(* Logix 5000 project; controller Program_Dampproduktion Emulate 5570 rev 32.11; software revision 32.02 *)

TASK MainTask (continuous, watchdog 500 ms) : Simulering
TASK Regulatorer (periodic, rate 100 ms, priority 10, watchdog 500 ms) : Regulator, Damp_Ventil_Regulering

MODULES
   Local : Emulate 5570 (ICP 3, rev 32.11)
END_MODULES

ADD_ON_INSTRUCTION Add_three_Numbers   (* revision 1.0 *)
VAR_INPUT
   nr1 : REAL; {required}
   nr2 : REAL; {required}
   nr3 : REAL; {required}
END_VAR
VAR_OUTPUT
   nr4 : REAL; {access Read Only, required}
END_VAR
VAR
   ADD_01 : FBD_MATH; {access None}
   ADD_02 : FBD_MATH; {access None}
   __lCF223809C1E0D70E : REAL; {access None}
   __l2841EC67DFDD29AE : REAL; {access None}
   __l253A293BB21A6975 : REAL; {access None}
END_VAR

ROUTINE Logic   (* function block diagram *)
   SHEET 1
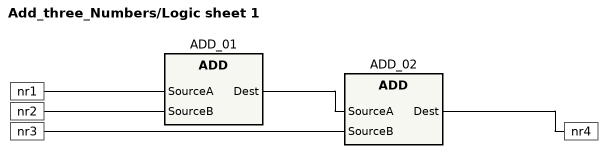
   ADD_01 : ADD(SourceA := nr1, SourceB := nr2);
   ADD_02 : ADD(SourceA := ADD_01.Dest, SourceB := nr3);
   nr4 := ADD_02.Dest;
END_ROUTINE
END_ADD_ON_INSTRUCTION

ADD_ON_INSTRUCTION DampProces   (* revision 1.0, vendor JPJohansen  *)
// Til obligatorisk opgave 1 - PA3
// Revision note:
// ændringer på dødtid og tidskonstant samt navn. den
VAR_INPUT
   belastning : REAL;
   DeadTime : REAL := 2.0;   // Dødtid 0.1 til 1.99 sek.
   Tidskonstant : REAL := 20.0;   // Tidskonstant i LeadLag 0.1 til 40.0 sek
END_VAR
VAR_OUTPUT
   PV : REAL; {access Read Only, required}
END_VAR
VAR_INPUT
   CV : REAL; {required}
END_VAR
VAR
   DEDT_01 : DEADTIME := (Deadtime := 1.0, Gain := 1.0, RTSTime := 1);
   ADD_01 : FBD_MATH;
   LDLG_01 : LEAD_LAG := (Lag := 20.0, Gain := 1.0, RTSTime := 1);
   HLL_01 : HL_LIMIT := (HighLimit := 100.0);
   SCL_01 : SCALE := (InRawMax := 100.0, InEUMax := 15.0, Limiting := 1); {access None}
   SCL_02 : SCALE := (InRawMax := 100.0, InEUMax := -100.0, Limiting := 1); {access None}
   StorageA : REAL[200]; {access None}
   SCL_03 : SCALE := (InRawMax := 100.0, InEUMin := 100.0, Limiting := 1); {access None}
   __lBFE748FCFA657C66 : REAL; {access None}
   __l111F0F8E6DFC85BE : REAL; {access None}
END_VAR

ROUTINE Logic   (* function block diagram *)
   SHEET 1
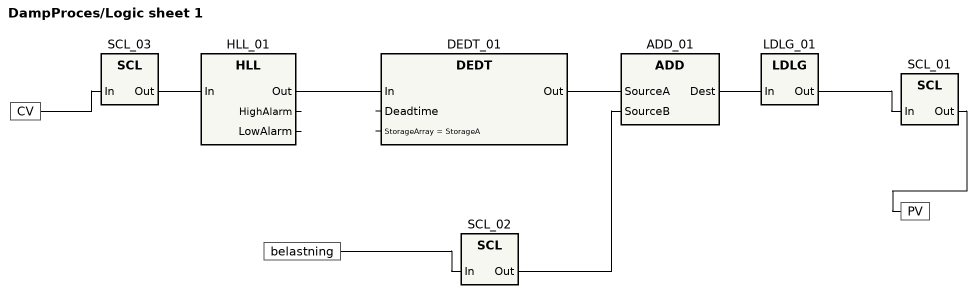
   SCL_03 : SCL(In := CV);
   HLL_01 : HLL(In := SCL_03.Out);   // unwired pins: HighAlarm LowAlarm
   DEDT_01 : DEDT(In := HLL_01.Out, StorageArray := StorageA);   // unwired pins: Deadtime
   SCL_02 : SCL(In := belastning);
   ADD_01 : ADD(SourceA := DEDT_01.Out, SourceB := SCL_02.Out);
   LDLG_01 : LDLG(In := ADD_01.Dest);
   SCL_01 : SCL(In := LDLG_01.Out);
   PV := SCL_01.Out;
END_ROUTINE
END_ADD_ON_INSTRUCTION

ADD_ON_INSTRUCTION Elektrodekammer   (* revision 1.0 *)
VAR_INPUT
   CV_Ind : REAL; {required}
END_VAR
VAR_OUTPUT
   PV_vandhojde : REAL; {access Read Only, required}
END_VAR
VAR_INPUT
   Belastning : REAL; {visible}
END_VAR
VAR
   LDLG_01 : LEAD_LAG := (Lag := 15.0, Gain := 1.4, RTSTime := 1); {access None}
   SUB_01 : FBD_MATH; {access None}
   DEDT_01 : DEADTIME := (Deadtime := 1.5, Gain := 1.5, RTSTime := 1); {access None}
   SCL_01 : SCALE := (InRawMax := 100.0, InEUMax := 100.0, Limiting := 1); {access None}
   SCL_02 : SCALE := (InRawMax := 100.0, InEUMax := 100.0, Limiting := 1); {access None}
   LDLG_02 : LEAD_LAG := (Lag := 10.0, Gain := 1.0, RTSTime := 1); {access None}
   Lag : REAL := 6.5; {access None}
   Gain_2 : REAL := 1.4; {access None}
   DeadTime : REAL := 0.5; {access None}
   Gain_1 : REAL := 0.9; {access None}
   StoreE : REAL[200]; {access None}
   __lBBB61524A4CF2047 : REAL; {access None}
   __l4C9B70D5358FCD80 : REAL; {access None}
   __lBCA77EE58B9857CC : REAL; {access None}
   __l311EF888CEB54C2F : REAL; {access None}
   __l26B57578D4CD21A6 : REAL; {access None}
   __l8BCF7D00DE459D5C : REAL; {access None}
END_VAR

ROUTINE Logic   (* function block diagram *)
   SHEET 1
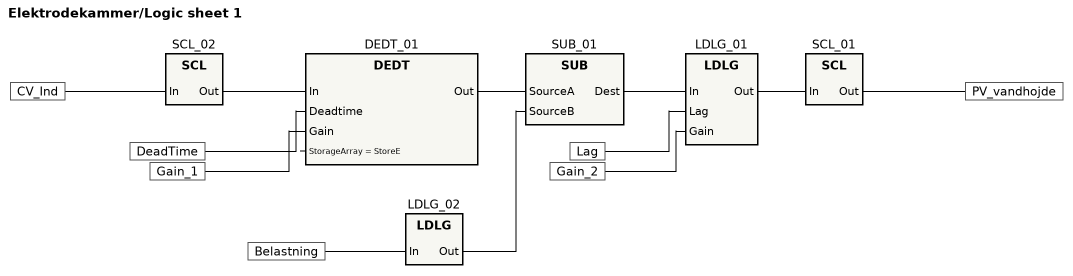
   SCL_02 : SCL(In := CV_Ind);
   DEDT_01 : DEDT(In := SCL_02.Out, Deadtime := DeadTime, Gain := Gain_1, StorageArray := StoreE);
   LDLG_02 : LDLG(In := Belastning);
   SUB_01 : SUB(SourceA := DEDT_01.Out, SourceB := LDLG_02.Out);
   LDLG_01 : LDLG(In := SUB_01.Dest, Lag := Lag, Gain := Gain_2);
   SCL_01 : SCL(In := LDLG_01.Out);
   PV_vandhojde := SCL_01.Out;
END_ROUTINE
END_ADD_ON_INSTRUCTION

ADD_ON_INSTRUCTION Foedevandskammer   (* revision 1.0 *)
VAR_INPUT
   CV_Ind : REAL; {required}
   Belastning : REAL; {visible}
END_VAR
VAR_OUTPUT
   PV_vandhojde : REAL; {access Read Only, required}
END_VAR
VAR
   LDLG_01 : LEAD_LAG := (Lag := 15.0, Gain := 1.4, RTSTime := 1); {access None}
   SUB_01 : FBD_MATH; {access None}
   DEDT_01 : DEADTIME := (Deadtime := 1.5, Gain := 1.5, RTSTime := 1); {access None}
   SCL_01 : SCALE := (InRawMax := 100.0, InEUMax := 100.0, Limiting := 1); {access None}
   SCL_02 : SCALE := (InRawMax := 100.0, InEUMax := 150.0, Limiting := 1); {access None}
   LDLG_02 : LEAD_LAG := (Lag := 10.0, Gain := 1.0, RTSTime := 1); {access None}
   DeadTime : REAL := 1.0; {access None}
   Gain_1 : REAL := 1.1; {access None}
   Lag : REAL := 8.0; {access None}
   Gain_2 : REAL := 1.2; {access None}
   StoreF : REAL[200]; {access None}
   __l47B9F860FB7F34CC : REAL; {access None}
   __lBCEEC7B2562564CC : REAL; {access None}
   __l8BD366BFA30A9B21 : REAL; {access None}
   __l726FB40F300CE841 : REAL; {access None}
   __l213C2E7ECA7368D6 : REAL; {access None}
   __l53F5B97CD43989B2 : REAL; {access None}
END_VAR

ROUTINE Logic   (* function block diagram *)
   SHEET 1
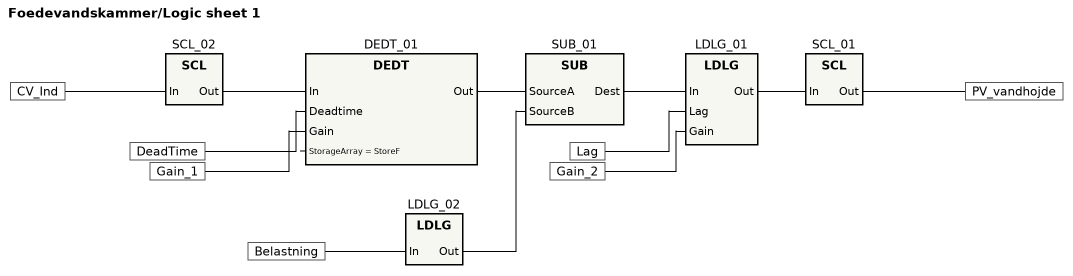
   SCL_02 : SCL(In := CV_Ind);
   DEDT_01 : DEDT(In := SCL_02.Out, Deadtime := DeadTime, Gain := Gain_1, StorageArray := StoreF);
   LDLG_02 : LDLG(In := Belastning);
   SUB_01 : SUB(SourceA := DEDT_01.Out, SourceB := LDLG_02.Out);
   LDLG_01 : LDLG(In := SUB_01.Dest, Lag := Lag, Gain := Gain_2);
   SCL_01 : SCL(In := LDLG_01.Out);
   PV_vandhojde := SCL_01.Out;
END_ROUTINE
END_ADD_ON_INSTRUCTION

ADD_ON_INSTRUCTION Invers_Direkte   (* revision 1.0 *)
VAR_INPUT
   PV : REAL; {required}
   SP : REAL; {required}
END_VAR
VAR_OUTPUT
   fejl_e : REAL; {access None, visible}
END_VAR
VAR_INPUT
   Invers_Direkte : BOOL; {access None, required}
END_VAR
VAR
   SUB_01 : FBD_MATH; {access None}
   SUB_02 : FBD_MATH; {access None}
   SEL_01 : SELECT; {access None}
   Invers : FBD_MATH; {access None}
   Direkte : FBD_MATH; {access None}
   __l92E14D13FB7A9B28 : BOOL; {access None}
   __l5E902B71B1A53267 : REAL; {access None}
   __lFF6ACCDBAA981339 : REAL; {access None}
END_VAR

ROUTINE Logic   (* function block diagram *)
   SHEET 1
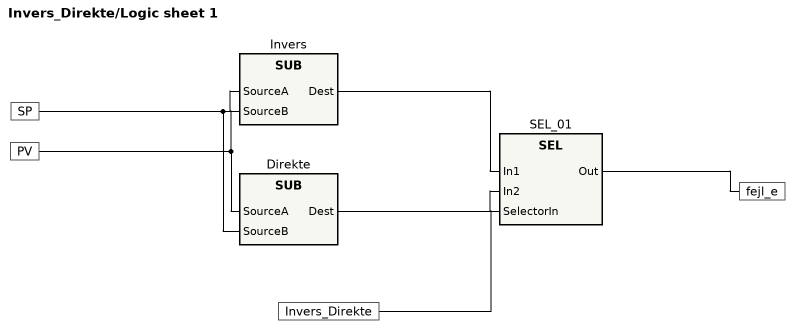
   Invers : SUB(SourceA := SP, SourceB := PV);
   Direkte : SUB(SourceA := PV, SourceB := SP);
   SEL_01 : SEL(In1 := Invers.Dest, In2 := Direkte.Dest, SelectorIn := Invers_Direkte);
   fejl_e := SEL_01.Out;
END_ROUTINE
END_ADD_ON_INSTRUCTION

ADD_ON_INSTRUCTION Kondenstank   (* revision 1.0, vendor Mr.Helgason *)
// Simulering af et kondenstank
// Help:
// *********************************
// Simulering af Vandmodeller
// *********************************
// Input:
// CV_in =  CV (Control Value) fra regulator 0-100% . REAL
// Belastning = Bruger indstiller 0 - 100%.  REAL
// Output:
// PV_vandhojde = Fra Level transmitter 0-100%. REAL
VAR_INPUT
   Belastning : REAL; {required}   // Belasting 0 - 100%
   CV_Ind : REAL; {required}   // 0 - 100%
END_VAR
VAR_OUTPUT
   PV_vandhojde : REAL; {access Read Only, required}   // 0 - 100%
END_VAR
VAR
   LDLG_01 : LEAD_LAG := (Lag := 15.0, Gain := 1.4, RTSTime := 1); {access None}
   SUB_01 : FBD_MATH; {access None}
   DEDT_01 : DEADTIME := (Deadtime := 1.5, Gain := 1.5, RTSTime := 1); {access None}
   DeadTime : REAL := 2.0; {access None}
   Store : REAL[200]; {access None}
   SCL_01 : SCALE := (InRawMax := 100.0, InEUMax := 100.0, Limiting := 1); {access None}
   SCL_02 : SCALE := (InRawMax := 100.0, InEUMax := 150.0, Limiting := 1); {access None}
   Gain_1 : REAL := 1.4; {access None}
   Lag : REAL := 15.0; {access None}
   Gain_2 : REAL := 1.2; {access None}
   LDLG_02 : LEAD_LAG := (Lag := 10.0, Gain := 1.0, RTSTime := 1); {access None}
   __l770FDFE62A3820F0 : REAL; {access None}
   __l2251F834FE043185 : REAL; {access None}
   __l3FFF9E27A9364976 : REAL; {access None}
   __lB3381F195010FDBE : REAL; {access None}
   __lEBAC3B9CE4C94A7F : REAL; {access None}
   __l23F97D3D6AB6734A : REAL; {access None}
END_VAR

ROUTINE Logic   (* function block diagram *)
   SHEET 1
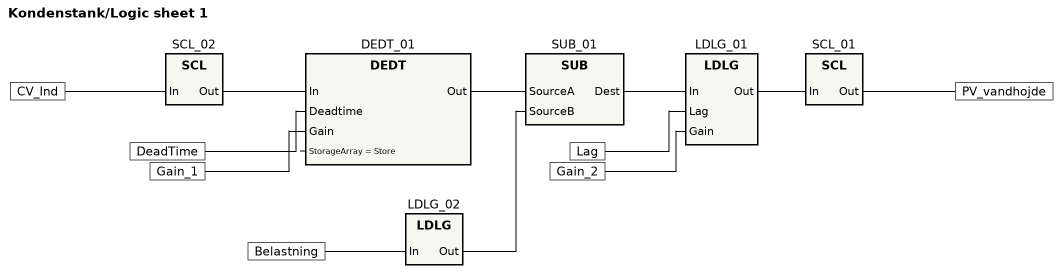
   SCL_02 : SCL(In := CV_Ind);
   DEDT_01 : DEDT(In := SCL_02.Out, Deadtime := DeadTime, Gain := Gain_1, StorageArray := Store);
   LDLG_02 : LDLG(In := Belastning);
   SUB_01 : SUB(SourceA := DEDT_01.Out, SourceB := LDLG_02.Out);
   LDLG_01 : LDLG(In := SUB_01.Dest, Lag := Lag, Gain := Gain_2);
   SCL_01 : SCL(In := LDLG_01.Out);
   PV_vandhojde := SCL_01.Out;
END_ROUTINE
END_ADD_ON_INSTRUCTION

ADD_ON_INSTRUCTION PID_regulator   (* revision 1.0 *)
VAR_INPUT
   SP : REAL; {access None, visible}
   PV : REAL; {access None, visible}
   Kp : REAL; {access None, visible}
   Ki : REAL; {access None, visible}
   Kd : REAL; {visible}
   U0 : REAL; {visible}
   U_man : REAL; {visible}
END_VAR
VAR_OUTPUT
   CV : REAL; {access Read Only, visible}
END_VAR
VAR_INPUT
   Invers_Direkte : BOOL; {access None, visible}
   Manuel_Auto : BOOL; {access None, visible}
   Zero_Ki : BOOL; {access None, visible}
END_VAR
VAR
   Add_three_Numbers_01 : Add_three_Numbers; {access None}
   Invers_Direkte_01 : Invers_Direkte; {access None}
   ADD_02 : FBD_MATH := (SourceA := 23.71752, Dest := 23.71752);
   DERV_01 : DERIVATIVE := (Gain := 5.0, RTSTime := 1, DeltaT := 0.1);
   INTG_01 : INTEGRATOR := (IGain := 4.0, HighLimit := 100.0, LowLimit := -100.0, RTSTime := 1, Out := 23.717138, DeltaT := 0.1);
   MUL_01 : FBD_MATH := (SourceB := 21.5);
   SEL_01 : SELECT;
   __l35FACD2691BF9949 : BOOL; {access None}
   __l9AC34CD4567C7C91 : REAL; {access None}
   __l01C926D5A08911AD : REAL; {access None}
   __l6354659A893A8F7F : REAL; {access None}
   __lF3243DCB1CB2B689 : BOOL; {access None}
   __l57A006EB2D259F2F : REAL; {access None}
   __l0F661682E7B60D3B : REAL; {access None}
   __l4E463AF5AF817CD4 : REAL; {access None}
   __lF1C43E32920F558F : REAL; {access None}
   __lE8A2B3305E3A9387 : BOOL; {access None}
END_VAR

ROUTINE Logic   (* function block diagram *)
   SHEET 1
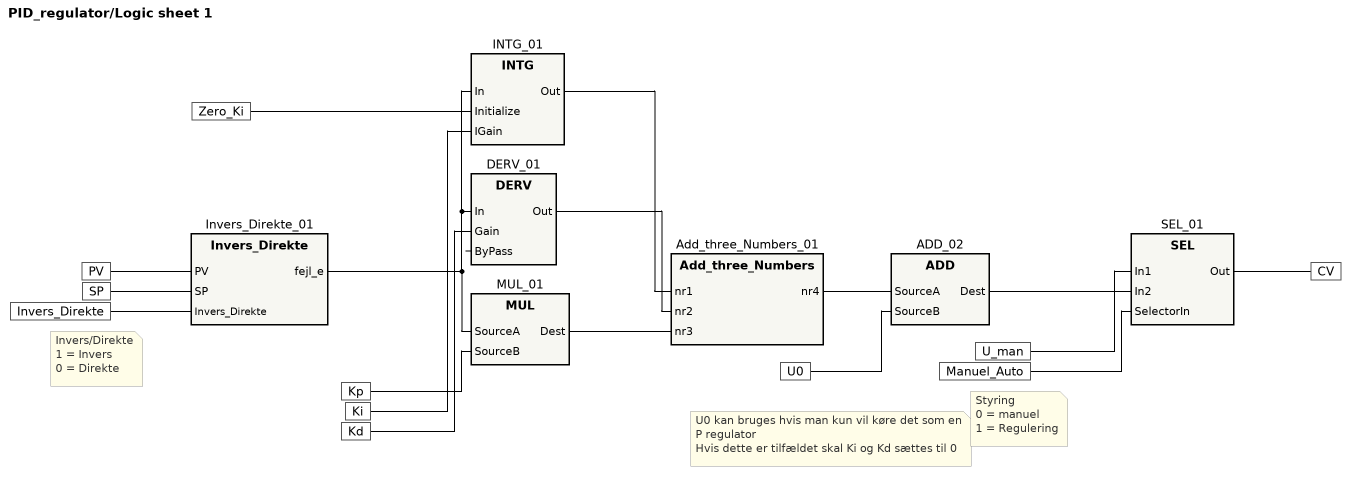
   // Invers/Direkte
   // 1 = Invers
   // 0 = Direkte
   Invers_Direkte_01 : Invers_Direkte(PV := PV, SP := SP, Invers_Direkte := Invers_Direkte);
   INTG_01 : INTG(In := Invers_Direkte_01.fejl_e, Initialize := Zero_Ki, IGain := Ki);
   DERV_01 : DERV(In := Invers_Direkte_01.fejl_e, Gain := Kd);   // unwired pins: ByPass
   MUL_01 : MUL(SourceA := Invers_Direkte_01.fejl_e, SourceB := Kp);
   Add_three_Numbers_01 : Add_three_Numbers(nr1 := INTG_01.Out, nr2 := DERV_01.Out, nr3 := MUL_01.Dest);
   // U0 kan bruges hvis man kun vil køre det som en
   // P regulator
   // Hvis dette er tilfældet skal Ki og Kd sættes til 0
   ADD_02 : ADD(SourceA := Add_three_Numbers_01.nr4, SourceB := U0);
   // Styring
   // 0 = manuel
   // 1 = Regulering
   SEL_01 : SEL(In1 := U_man, In2 := ADD_02.Dest, SelectorIn := Manuel_Auto);
   CV := SEL_01.Out;
END_ROUTINE
END_ADD_ON_INSTRUCTION

VAR_GLOBAL   (* controller tags *)
   AT_DP_kaska : PIDE_AUTOTUNE;
   CP_4 : REAL;
   Damp_CV : REAL;
   E1_E2 : BOOL;
   Elektrode : BOOL;
   initialize : BOOL;
   initValue : REAL;
   Kd : REAL;
   Ki : REAL;
   Ki_damp : REAL;
   Kp_damp : REAL;
   OpenValue_V3 : REAL := 9.0;
   PT_3 : REAL;
   SP : REAL;
   SP_Damp : REAL := 9.5;
   Tryk_stigning : REAL;
   V3 : REAL;
END_VAR

PROGRAM Damp_Ventil_Regulering   (* main routine Regulator *)
VAR
   BNOT_01 : FBD_BOOLEAN_NOT := (Out := 1);
   GRT_01 : FBD_COMPARE := (SourceA := 1.1071618e-05, SourceB := 9.0);
   PID_regulator_01 : PID_regulator := (SP := 9.5, PV := 1.1071618e-05, Kp := 60.0, Ki := 7.0, CV := -569.9993, Invers_Direkte := 1, Manuel_Auto := 1, Zero_Ki := 1);
   SEL_01 : SELECT;
END_VAR

ROUTINE Regulator   (* function block diagram *)
   SHEET 1
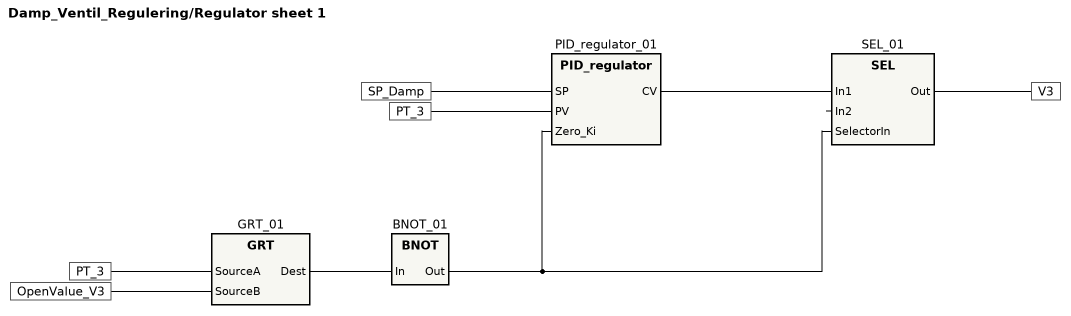
   GRT_01 : GRT(SourceA := PT_3, SourceB := OpenValue_V3);
   BNOT_01 : BNOT(In := GRT_01.Dest);
   PID_regulator_01 : PID_regulator(SP := SP_Damp, PV := PT_3, Zero_Ki := BNOT_01.Out);
   SEL_01 : SEL(In1 := PID_regulator_01.CV, SelectorIn := BNOT_01.Out);   // unwired pins: In2
   V3 := SEL_01.Out;
END_ROUTINE
END_PROGRAM

PROGRAM Regulator   (* main routine Main *)
VAR
   FT4 : REAL;
   Kd_DP_flow_kaska : REAL;
   Ki_damp_kaska : REAL;
   Ki_DP_flow_kaska : REAL;
   Kp_damp_kaska : REAL;
   Kp_DP_flow_kaska : REAL;
   Level_SP_kW : REAL;
   LT_4 : REAL;
   PIDE_01 : PID_ENHANCED := (PVEUMax := 100.0, SPHLimit := 100.0, RatioProg := 1.0, RatioOper := 1.0, RatioHLimit := 1.0, RatioLLimit := 1.0, CVEUMax := 100.0, CVHLimit := 100.0, PVEDerivative := 1, RTSTime := 1);
   PIDE_02 : PID_ENHANCED := (PVEUMax := 100.0, SPHLimit := 100.0, RatioProg := 1.0, RatioOper := 1.0, RatioHLimit := 1.0, RatioLLimit := 1.0, CVEUMax := 100.0, CVHLimit := 100.0, PVEDerivative := 1, RTSTime := 1);
   PIDE_03 : PID_ENHANCED := (PVEUMax := 100.0, SPHLimit := 100.0, RatioProg := 1.0, RatioOper := 1.0, RatioHLimit := 1.0, RatioLLimit := 1.0, CVEUMax := 100.0, CVHLimit := 100.0, PVEDerivative := 1, RTSTime := 1);
   SCL_01 : SCALE;
   U_damp_manuel : REAL;
END_VAR

ROUTINE Kaskaderegulator_Dampproduktion   (* function block diagram *)
   SHEET 1
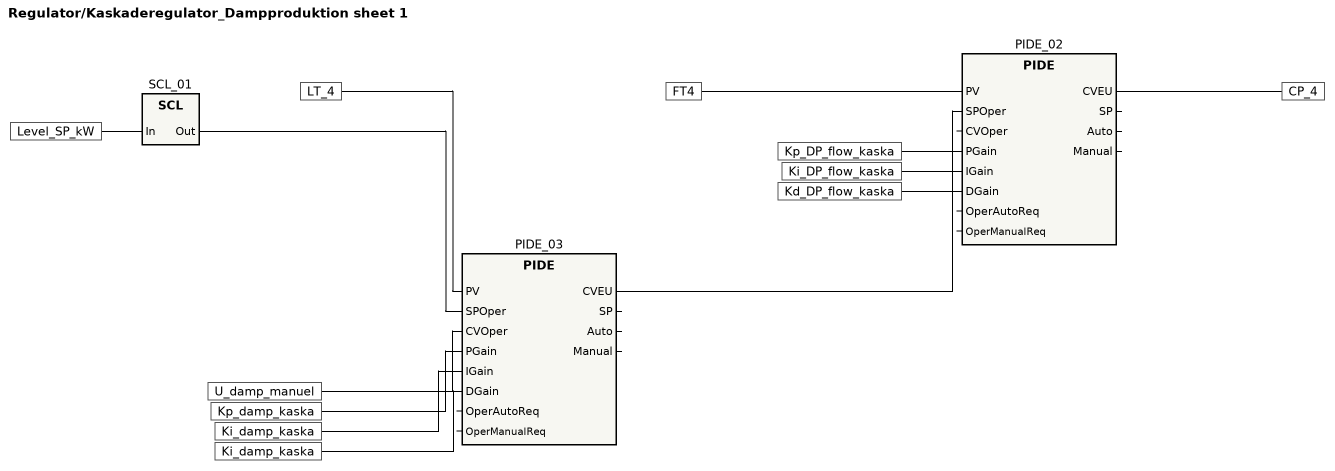
   SCL_01 : SCL(In := Level_SP_kW);
   PIDE_03 : PIDE(PV := LT_4, SPOper := SCL_01.Out, CVOper := U_damp_manuel, PGain := Kp_damp_kaska, IGain := Ki_damp_kaska, DGain := Ki_damp_kaska);   // unwired pins: OperAutoReq OperManualReq SP Auto Manual
   PIDE_02 : PIDE(PV := FT4, SPOper := PIDE_03.CVEU, PGain := Kp_DP_flow_kaska, IGain := Ki_DP_flow_kaska, DGain := Kd_DP_flow_kaska);   // unwired pins: CVOper OperAutoReq OperManualReq SP Auto Manual
   CP_4 := PIDE_02.CVEU;
END_ROUTINE

ROUTINE Main   (* ladder *)
END_ROUTINE

ROUTINE Niveauregulator_Dampproduktion   (* function block diagram *)
   SHEET 1
END_ROUTINE
END_PROGRAM

PROGRAM Simulering   (* main routine Main *)
VAR
   DampProces_01 : DampProces := (DeadTime := 2.0, Tidskonstant := 20.0);
   EQU_01 : FBD_COMPARE;
   SCL_01 : SCALE := (InRawMax := 30000.0, InEUMin := 100.0, Limiting := 1, Out := 100.0);
   SEL_01 : SELECT;
   TONR_01 : FBD_TIMER := (PRE := 30000);
END_VAR

ROUTINE DampProces_Simulering   (* function block diagram *)
   SHEET 1
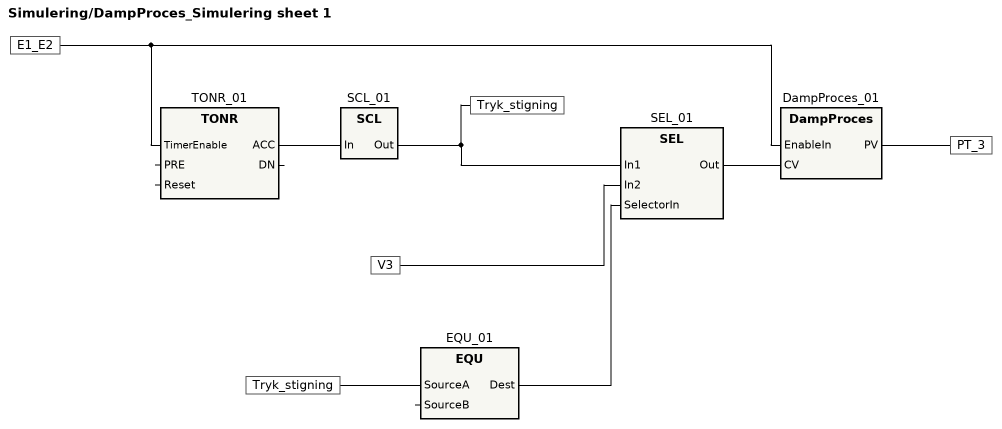
   TONR_01 : TONR(TimerEnable := E1_E2);   // unwired pins: PRE Reset DN
   SCL_01 : SCL(In := TONR_01.ACC);
   EQU_01 : EQU(SourceA := Tryk_stigning);   // unwired pins: SourceB
   Tryk_stigning := SCL_01.Out;
   SEL_01 : SEL(In1 := SCL_01.Out, In2 := V3, SelectorIn := EQU_01.Dest);
   DampProces_01 : DampProces(EnableIn := E1_E2, CV := SEL_01.Out);
   PT_3 := DampProces_01.PV;
END_ROUTINE

ROUTINE Elektrodekammer   (* function block diagram *)
   SHEET 1
END_ROUTINE

ROUTINE Foedevandskammer   (* function block diagram *)
   SHEET 1
END_ROUTINE

ROUTINE Kondenstank   (* function block diagram *)
   SHEET 1
END_ROUTINE

ROUTINE Main   (* ladder *)
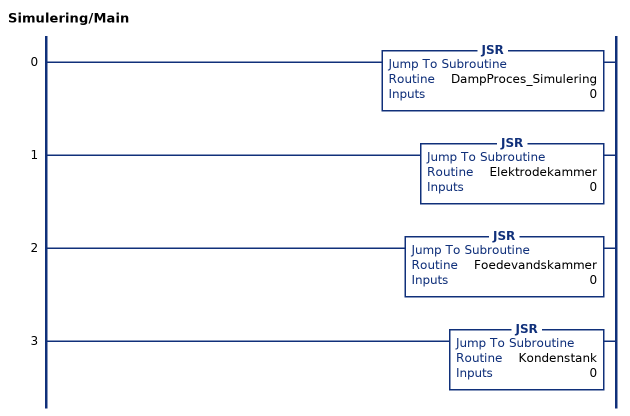
   0: JSR(DampProces_Simulering,0);
   1: JSR(Elektrodekammer,0);
   2: JSR(Foedevandskammer,0);
   3: JSR(Kondenstank,0);
END_ROUTINE
END_PROGRAM
